// Mitsubishi GX Works2 project: AND ESTRUTURADO   PLC: Q03UDV

// task Task_01 (event TRUE, interval 0, priority 31): POU_01

PROGRAM POU_01
VAR
  mo : BOOL;
  CTD_1 : CTD;
  CTU_1 : CTU;
  CTUD_1 : CTUD;
  TP_1 : TP;
  TON_1 : TON;
  TOF_1 : TOF;
  tp1 : TIME;
  ton1 : TIME;
  time_off : TIME;
  time_on : TIME;
  fbBlinker_1 : fbBlinker;
  fbBlinker_2 : fbBlinker;
END_VAR
(* structured ladder/FBD written out as ST: instructions are called as NAME(EN, inputs, outputs); _pN, _eN, _tN stand for wires *)
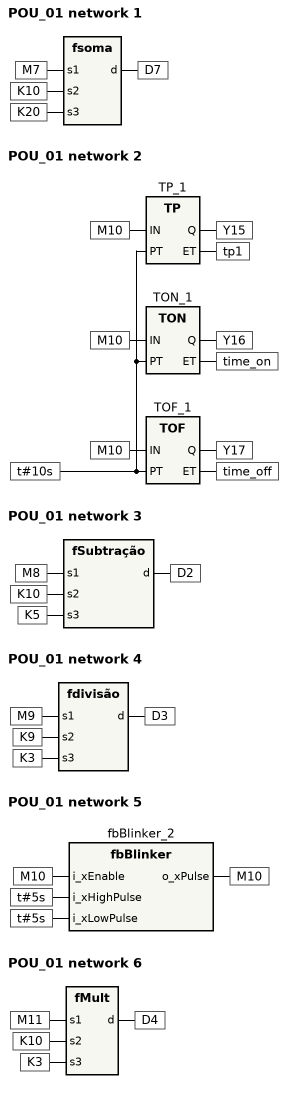
(* network 1 *)
D7 := fsoma(M7, K10, K20);
(* network 2 *)
TP_1(IN := M10, PT := t#10s, Q => Y15, ET => tp1);
TON_1(IN := M10, PT := t#10s, Q => Y16, ET => time_on);
TOF_1(IN := M10, PT := t#10s, Q => Y17, ET => time_off);
(* network 3 *)
D2 := fSubtração(M8, K10, K5);
(* network 4 *)
D3 := fdivisão(M9, K9, K3);
(* network 5 *)
fbBlinker_2(i_xEnable := M10, i_xHighPulse := t#5s, i_xLowPulse := t#5s, o_xPulse => M10);
(* network 6 *)
D4 := fMult(M11, K10, K3);
END_PROGRAM

FUNCTION fsoma
VAR_INPUT
  i_xHabilitar : BOOL;
  i_iElemento1 : INT;
  i_iElemento2 : INT;
END_VAR
(* structured ladder/FBD written out as ST: instructions are called as NAME(EN, inputs, outputs); _pN, _eN, _tN stand for wires *)
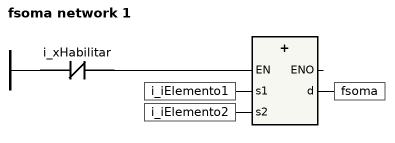
(* network 1 *)
+(NOT i_xHabilitar, i_iElemento1, i_iElemento2, fsoma);
END_FUNCTION

FUNCTION fSubtração
VAR_INPUT
  i_xHabilitarSub : BOOL;
  i_iElemento1 : INT;
  i_iElemento2 : INT;
END_VAR
(* structured ladder/FBD written out as ST: instructions are called as NAME(EN, inputs, outputs); _pN, _eN, _tN stand for wires *)
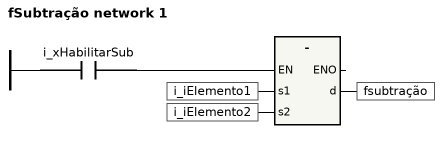
(* network 1 *)
-(i_xHabilitarSub, i_iElemento1, i_iElemento2, fsubtração);
END_FUNCTION

FUNCTION fdivisão
VAR_INPUT
  i_xHabilitarDiv : BOOL;
  i_iElemento1 : INT;
  i_iElemento2 : INT;
END_VAR
(* structured ladder/FBD written out as ST: instructions are called as NAME(EN, inputs, outputs); _pN, _eN, _tN stand for wires *)
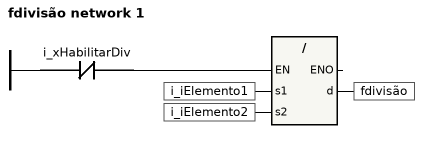
(* network 1 *)
/(NOT i_xHabilitarDiv, i_iElemento1, i_iElemento2, fdivisão);
END_FUNCTION

FUNCTION_BLOCK fbBlinker
VAR_INPUT
  i_xEnable : BOOL;
  i_xHighPulse : TIME;
  i_xLowPulse : TIME;
END_VAR
VAR_OUTPUT
  o_xPulse : BOOL;
END_VAR
VAR
  fb_TimerHigh : TP;
  fb_TimerLow : TOF;
  xAuxiliar : BOOL;
END_VAR
(* structured ladder/FBD written out as ST: instructions are called as NAME(EN, inputs, outputs); _pN, _eN, _tN stand for wires *)
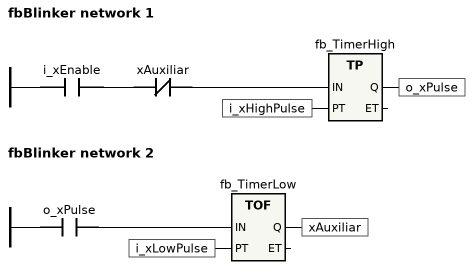
(* network 1 *)
fb_TimerHigh(IN := i_xEnable AND NOT xAuxiliar, PT := i_xHighPulse, Q => o_xPulse);
(* network 2 *)
fb_TimerLow(IN := o_xPulse, PT := i_xLowPulse, Q => xAuxiliar);
END_FUNCTION_BLOCK

FUNCTION fMult
VAR_INPUT
  i_xHabilitarMult : BOOL;
  i_iElemento1 : INT;
  i_iElemento2 : INT;
END_VAR
(* structured ladder/FBD written out as ST: instructions are called as NAME(EN, inputs, outputs); _pN, _eN, _tN stand for wires *)
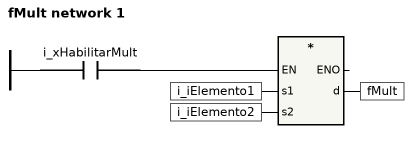
(* network 1 *)
*(i_xHabilitarMult, i_iElemento1, i_iElemento2, fMult);
END_FUNCTION
